{attribute 'reflection'}
FUNCTION_BLOCK INTERNAL FINAL FB_Snappy_Tests EXTENDS TcUnit.FB_TestSuite
VAR_INPUT
END_VAR
VAR_OUTPUT
END_VAR
VAR
	{attribute 'instance-path'} 
    {attribute 'noinit'} 
	sTestName			: T_MaxString;
END_VAR

TEST(sTestName);

ShouldInitializeDefaultsSuccessfully();
//Debug();
TEST_FINISHED_NAMED(sTestName);

METHOD PRIVATE Debug
VAR_INST
	
	hr		: HRESULT;		
	fbAdapter : FB_TcUnitAdapter;
END_VAR

TEST('Test some stuff');

// ARRANGE

// ACT and ASSERT
hr := fbAdapter.Verify(anyArg:= _AppInfo);

IF NOT PENDING(hr) THEN
	TEST_FINISHED_NAMED('Test some stuff');
END_IF;
END_METHOD

METHOD PRIVATE ShouldInitializeDefaultsSuccessfully
VAR_INST
	fbSUT		: FB_Snappy;
	hr			: HRESULT;	
END_VAR

TEST('ShuldInitializeDefaultsSuccessfully');

// Arrange
// Act
hr := fbSUT.Configure().UseDefaults().WithoutTestFramework(sTestSuiteName:='MyTestSuite', sTestName:='MyTestName').Build();

// Assert

AssertEquals_DINT(Expected:= S_OK,
				Actual:= hr,
				Message:= 'Expected HRESULT=S_OK');


TEST_FINISHED();
END_METHOD

METHOD PRIVATE Shouldxxx
VAR_INST
	hr		: HRESULT;	
END_VAR

TEST('Shouldxxx');

// Arrange

// Act

// Assert
AssertEquals_DINT(Expected:= S_OK,
					Actual:= hr,
					Message:= 'Expected HRESULT=S_OK');

TEST_FINISHED();
END_METHOD

END_FUNCTION_BLOCK

(* stored: Version 1.1.0.1, ProductVersion 3.1.4026.18
   POU FB_Snappy_Tests: Id {4ce24020-c3c6-49c2-8321-f54e613b89e8}, SpecialFunc None
   Method Debug: Id {e1697c70-17fa-4f58-ac00-58cd8276447b}
   Method ShouldInitializeDefaultsSuccessfully: Id {b0bee8e3-0ce4-4d03-b00a-9672e47157fa}
   Method Shouldxxx: Id {2ed23d4e-8e1b-49bf-ad1c-93e42dfcde7b} *)
